(* IEC 61131-3 sources: CodesysTest/export/SX_1195.dev/Plc Logic/Application/PRJ Specific/1195 Testing, 2 files *)

(* ---- sctMotionProfile.dut.st ---- *)
(*#-#-#-#-#-#-#-#-#-#---Declaration---#-#-#-#-#-#-#-#-#-#-#-#-#*)

TYPE sctMotionProfile :
STRUCT
	velocity : REAL;
	acceleration : REAL;
	deceleration : REAL;
	position : REAL;
	minPosition : REAL;
	maxPosition : REAL;
	current : REAL;
END_STRUCT
END_TYPE

(* ---- F_EtherCatSlaveCommsRunning.pou.st ---- *)
(*#-#-#-#-#-#-#-#-#-#---Declaration---#-#-#-#-#-#-#-#-#-#-#-#-#*)

FUNCTION F_EtherCatSlaveCommsRunning : BOOL
VAR_INPUT
	state : IoDrvEthercatLib.ETC_SLAVE_STATE;
END_VAR
VAR
END_VAR
(*#-#-#-#-#-#-#-#-#-#---Implementation---#-#-#-#-#-#-#-#-#-#-#-#-#*)

F_EtherCatSlaveCommsRunning := NOT (state = IoDrvEthercatLib.ETC_SLAVE_STATE.ETC_SLAVE_INIT);
